% RSLogix 500 project Intro to Automation Hands On Final.RSS, saved by version 10.00.00.00 %
PROJECT "ML06B"    % processor: Bul.1763 MicroLogix 1100 Series B %

PROGRAM FILES
  LAD 2   5 rungs

DATA FILES
  O0 OUTPUT  4 elements  % Output 4 %
  I1 INPUT  6 elements
  S2 STATUS  66 elements
  B3 BINARY  1 elements
  T4 TIMER  1 elements
  C5 COUNTER  1 elements
  R6 CONTROL  1 elements
  N7 INTEGER  1 elements
  F8 FLOAT  1 elements

LADDER 2
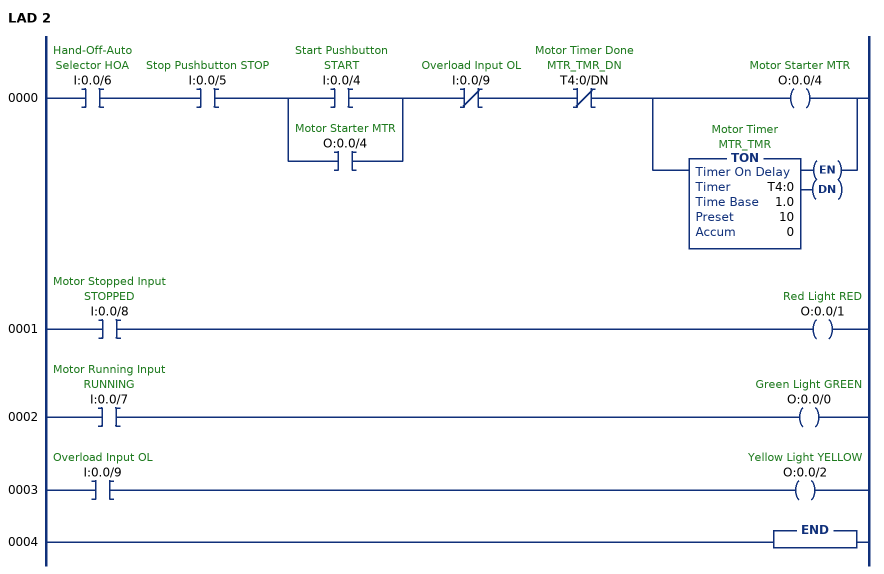
% Rung: 0 %
SOR XIC I:0.0/6 XIC I:0.0/5 BST XIC I:0.0/4 NXB XIC O:0.0/4 BND XIO I:0.0/9 XIO T4:0/DN BST OTE O:0.0/4 NXB TON T4:0 1.0 10 0 BND EOR
%   I:0.0/6  HOA  "Hand-Off-Auto Selector" %
%   I:0.0/5  STOP  "Stop Pushbutton" %
%   I:0.0/4  START  "Start Pushbutton" %
%   O:0.0/4  MTR  "Motor Starter" %
%   I:0.0/9  OL  "Overload Input" %
%   T4:0/DN  MTR_TMR_DN  "Motor Timer Done" %
%   T4:0  MTR_TMR  "Motor Timer" %
% Rung: 1 %
SOR XIC I:0.0/8 OTE O:0.0/1 EOR
%   I:0.0/8  STOPPED  "Motor Stopped Input" %
%   O:0.0/1  RED  "Red Light" %
% Rung: 2 %
SOR XIC I:0.0/7 OTE O:0.0/0 EOR
%   I:0.0/7  RUNNING  "Motor Running Input" %
%   O:0.0/0  GREEN  "Green Light" %
% Rung: 3 %
SOR XIC I:0.0/9 OTE O:0.0/2 EOR
%   I:0.0/9  OL  "Overload Input" %
%   O:0.0/2  YELLOW  "Yellow Light" %
% Rung: 4 %
SOR END EOR

OTHER DOCUMENTED ADDRESSES
  I:0.0  SEL_P1
  O:0.0/3  GRN_LT2  "Green Light 2"
  T4:0/EN  MTR_TMR_EN

DATA TABLE (non-zero values as saved)
DATA T4
% .PRE .ACC %
% T4:0 % 10 0
